TYPE ST_RecipeControl :
STRUCT
	iType					:INT;
	bCreate					:BOOL;
	bRefresh				:BOOL;
	bOpen					:BOOL;
	bClose					:BOOL;
	bDelete					:BOOL;
	iIndex					:INT;
	iList					:INT;
END_STRUCT
END_TYPE

(* stored: Version 1.1.0.1
   DUT ST_RecipeControl: Id {bcb743e8-a09e-48bc-be56-b4beb6a42032} *)
